// TIA Portal V20 export
TYPE "LBP_typeModeGroup"
TITLE = Mode group signals / Signaux groupe de modes de fonctionnement
// User data type for block LBP_ModeGroup [DB11] / Type de données utilisateur pour bloc LBP_ModeGroup [DB11]
   STRUCT
      A_AUTO : Bool;   // Operating mode AUTOMATIC / Mode AUTOMATIC
      A_MDA : Bool;   // Operating mode MDA / Mode MDA
      A_JOG : Bool;   // Operating mode JOG / Mode JOG
      f0_3 : Bool;
      A_MCDisable : Bool;   // Mode change disable / Désactiver changement mode de fonctionnement
      A_MGStop : Bool;   // Mode group stop / Groupe de modes de fonctionnement Arrêt
      A_MGStopASp : Bool;   // Mode group stop axes plus spindle / Groupe de modes de fonctionnement Arrêt axes et broche
      A_MGReset : Bool;   // Mode group reset / Groupe de modes de fonctionnement Reset
      A_TEACHIN : Bool;   // Machine function TEACH IN / Fonction machine TEACH IN
      A_REPOS : Bool;   // Machine function REPOS / Fonction machine REPOS
      A_REF : Bool;   // Machine function REF / Fonction machine REF
      f1_3 : Bool;
      f1_4 : Bool;
      f1_5 : Bool;
      A_SingleBlock_B : Bool;   // Single block type B / Bloc par bloc type B
      A_SingleBlock_A : Bool;   // Single block type A / Bloc par bloc type A
      A_INC1 : Bool;   // INC1
      A_INC10 : Bool;   // INC10
      A_INC100 : Bool;   // INC100
      A_INC1000 : Bool;   // INC1000
      A_INC10000 : Bool;   // INC10000
      A_INCVar : Bool;   // INC variable / Variable INC
      A_ContManTravel : Bool;   // Continuous manual travel / Mode manuel continu
      f2_7 : Bool;
      f3 : Byte;
      E_MMC_AUTO : Bool;   // HMI mode strobe AUTOMATIC / HMI mode Strobe AUTOMATIC
      E_MMC_MDA : Bool;   // HMI mode strobe MDA / HMI mode Strobe MDA
      E_MMC_JOG : Bool;   // HMI mode strobe JOG / HMI mode Strobe JOG
      f4_3 : Bool;
      f4_4 : Bool;
      f4_5 : Bool;
      f4_6 : Bool;
      f4_7 : Bool;
      E_MMC_TEACHIN : Bool;   // HMI machine function strobe TEACH IN / HMI Fonction machine Strobe TEACH IN
      E_MMC_REPOS : Bool;   // HMI machine function strobe REPOS / HMI Fonction machine Strobe REPOS
      E_MMC_REF : Bool;   // HMI machine function strobe REF / HMI Fonction machine Strobe REF
      f5_3 : Bool;
      f5_4 : Bool;
      f5_5 : Bool;
      f5_6 : Bool;
      f5_7 : Bool;
      E_AUTO : Bool;   // Active operating mode AUTOMATIC / Mode actif AUTOMATIC
      E_MDA : Bool;   // Active operating mode MDA / Mode actif MDA
      E_JOG : Bool;   // Active operating mode JOG / Mode actif JOG
      E_MGOK : Bool;   // Mode group ready / Groupe de modes de fonctionnement prêt
      E_MGreseted : Bool;   // Mode group reset performed / Groupe de modes de fonctionnement Reset effectué
      E_NCKintJOG : Bool;   // NCK internal JOG active / NCK JOG interne actif
      f6_6 : Bool;
      E_ChanReset : Bool;   // All channels in reset state / Tous les canaux en mode Reset
      E_TEACHIN : Bool;   // Active machine function TEACH IN / Fonction machine active TEACH IN
      E_REPOS : Bool;   // Active machine function REPOS / Fonction machine active REPOS
      E_REF : Bool;   // Active machine function REF / Fonction machine active REF
      f7_3 : Bool;
      f7_4 : Bool;
      f7_5 : Bool;
      f7_6 : Bool;
      f7_7 : Bool;
      E_INC1 : Bool;   // INC1
      E_INC10 : Bool;   // INC10
      E_INC100 : Bool;   // INC100
      E_INC1000 : Bool;   // INC1000
      E_INC10000 : Bool;   // INC10000
      E_INCVar : Bool;   // INC variable / Variable INC
      E_ContManTravelAct : Bool;   // Continuous manual travel active / Mode manuel continu actif
      f8_7 : Bool;
      f9 : Byte;
      E_HMI_INC1 : Bool;   // INC1 from HMI / INC1 depuis IHM
      E_HMI_INC10 : Bool;   // INC10 from HMI / INC10 depuis IHM
      E_HMI_INC100 : Bool;   // INC100 from HMI / INC100 depuis IHM
      E_HMI_INC1000 : Bool;   // INC1000 from HMI / INC1000 depuis IHM
      E_HMI_INC10000 : Bool;   // INC10000 from HMI / INC10000 depuis IHM
      E_HMI_INCVar : Bool;   // INC variable from HMI / Variable INC depuis IHM
      E_HMI_ContManTravel : Bool;   // Continuous manual travel active from HMI / Course manuelle continue active depuis IHM
      f10_7 : Bool;
      f11 : Byte;
      f12 : Array[12..19] of Byte;
      MG : Array[2..10] of Struct   // next mode group from DBB20, as before / groupe de mode suivant depuis DBB20, comme avant
         A_AUTO : Bool;   // Operating mode AUTOMATIC / Mode AUTOMATIC
         A_MDA : Bool;   // Operating mode MDA / Mode MDA
         A_JOG : Bool;   // Operating mode JOG / Mode JOG
         f0_3 : Bool;
         A_MCDisable : Bool;   // Mode change disable / Désactiver changement mode de fonctionnement
         A_MGStop : Bool;   // Mode group stop / Groupe de modes de fonctionnement Arrêt
         A_MGStopASp : Bool;   // Mode group stop axes plus spindle / Groupe de modes de fonctionnement Arrêt axes et broche
         A_MGReset : Bool;   // Mode group reset / Groupe de modes de fonctionnement Reset
         A_TEACHIN : Bool;   // Machine function TEACH IN / Fonction machine TEACH IN
         A_REPOS : Bool;   // Machine function REPOS / Fonction machine REPOS
         A_REF : Bool;   // Machine function REF / Fonction machine REF
         f1_3 : Bool;
         f1_4 : Bool;
         f1_5 : Bool;
         A_SingleBlock_B : Bool;   // Single block type B / Bloc par bloc type B
         A_SingleBlock_A : Bool;   // Single block type A / Bloc par bloc type A
         A_INC1 : Bool;   // INC1
         A_INC10 : Bool;   // INC10
         A_INC100 : Bool;   // INC100
         A_INC1000 : Bool;   // INC1000
         A_INC10000 : Bool;   // INC10000
         A_INCVar : Bool;   // INC variable / Variable INC
         A_ContManTravel : Bool;   // Continuous manual travel / Mode manuel continu
         f2_7 : Bool;
         f3 : Byte;
         E_MMC_AUTO : Bool;   // HMI mode strobe AUTOMATIC / HMI mode Strobe AUTOMATIC
         E_MMC_MDA : Bool;   // HMI mode strobe MDA / HMI mode Strobe MDA
         E_MMC_JOG : Bool;   // HMI mode strobe JOG / HMI mode Strobe JOG
         f4_3 : Bool;
         f4_4 : Bool;
         f4_5 : Bool;
         f4_6 : Bool;
         f4_7 : Bool;
         E_MMC_TEACHIN : Bool;   // HMI machine function strobe TEACH IN / HMI Fonction machine Strobe TEACH IN
         E_MMC_REPOS : Bool;   // HMI machine function strobe REPOS / HMI Fonction machine Strobe REPOS
         E_MMC_REF : Bool;   // HMI machine function strobe REF / HMI Fonction machine Strobe REF
         f5_3 : Bool;
         f5_4 : Bool;
         f5_5 : Bool;
         f5_6 : Bool;
         f5_7 : Bool;
         E_AUTO : Bool;   // Active operating mode AUTOMATIC / Mode actif AUTOMATIC
         E_MDA : Bool;   // Active operating mode MDA / Mode actif MDA
         E_JOG : Bool;   // Active operating mode JOG / Mode actif JOG
         E_MGOK : Bool;   // Mode group ready / Groupe de modes de fonctionnement prêt
         E_MGreseted : Bool;   // Mode group reset / Groupe de modes de fonctionnement Reset
         E_NCKintJOG : Bool;   // NCK internal JOG active / NCK JOG interne actif
         f6_6 : Bool;
         E_ChanReset : Bool;   // All channels in reset state / Tous les canaux en mode Reset
         E_TEACHIN : Bool;   // Active machine function TEACH IN / Fonction machine active TEACH IN
         E_REPOS : Bool;   // Active machine function REPOS / Fonction machine active REPOS
         E_REF : Bool;   // Active machine function REF / Fonction machine active REF
         f7_3 : Bool;
         f7_4 : Bool;
         f7_5 : Bool;
         f7_6 : Bool;
         f7_7 : Bool;
         E_INC1 : Bool;   // INC1
         E_INC10 : Bool;   // INC10
         E_INC100 : Bool;   // INC100
         E_INC1000 : Bool;   // INC1000
         E_INC10000 : Bool;   // INC10000
         E_INCVar : Bool;   // INC variable / Variable INC
         E_ContManTravelAct : Bool;   // Continuous manual travel active / Mode manuel continu actif
         f8_7 : Bool;
         f9 : Byte;
         E_HMI_INC1 : Bool;   // INC1 from HMI / INC1 depuis IHM
         E_HMI_INC10 : Bool;   // INC10 from HMI / INC10 depuis IHM
         E_HMI_INC100 : Bool;   // INC100 from HMI / INC100 depuis IHM
         E_HMI_INC1000 : Bool;   // INC1000 from HMI / INC1000 depuis IHM
         E_HMI_INC10000 : Bool;   // INC10000 from HMI / INC10000 depuis IHM
         E_HMI_INCVar : Bool;   // INC variable from HMI / Variable INC depuis IHM
         E_HMI_ContManTravel : Bool;   // Continuous manual travel active from HMI / Course manuelle continue active depuis IHM
         f10_7 : Bool;
         f11 : Byte;
         f12 : Array[12..19] of Byte;
      END_STRUCT;
   END_STRUCT;
   // // MG[3].A_AUTO : Operating mode AUTOMATIC / Mode AUTOMATIC
   // // MG[4].A_AUTO : Operating mode AUTOMATIC / Mode AUTOMATIC
   // // MG[5].A_AUTO : Operating mode AUTOMATIC / Mode AUTOMATIC
   // // MG[6].A_AUTO : Operating mode AUTOMATIC / Mode AUTOMATIC
   // // MG[7].A_AUTO : Operating mode AUTOMATIC / Mode AUTOMATIC
   // // MG[8].A_AUTO : Operating mode AUTOMATIC / Mode AUTOMATIC
   // // MG[9].A_AUTO : Operating mode AUTOMATIC / Mode AUTOMATIC
   // // MG[10].A_AUTO : Operating mode AUTOMATIC / Mode AUTOMATIC
   // // MG[3].A_MDA : Operating mode MDA / Mode MDA
   // // MG[4].A_MDA : Operating mode MDA / Mode MDA
   // // MG[5].A_MDA : Operating mode MDA / Mode MDA
   // // MG[6].A_MDA : Operating mode MDA / Mode MDA
   // // MG[7].A_MDA : Operating mode MDA / Mode MDA
   // // MG[8].A_MDA : Operating mode MDA / Mode MDA
   // // MG[9].A_MDA : Operating mode MDA / Mode MDA
   // // MG[10].A_MDA : Operating mode MDA / Mode MDA
   // // MG[3].A_JOG : Operating mode JOG / Mode JOG
   // // MG[4].A_JOG : Operating mode JOG / Mode JOG
   // // MG[5].A_JOG : Operating mode JOG / Mode JOG
   // // MG[6].A_JOG : Operating mode JOG / Mode JOG
   // // MG[7].A_JOG : Operating mode JOG / Mode JOG
   // // MG[8].A_JOG : Operating mode JOG / Mode JOG
   // // MG[9].A_JOG : Operating mode JOG / Mode JOG
   // // MG[10].A_JOG : Operating mode JOG / Mode JOG
   // // MG[3].A_MCDisable : Mode change disable / Désactiver changement mode de fonctionnement
   // // MG[4].A_MCDisable : Mode change disable / Désactiver changement mode de fonctionnement
   // // MG[5].A_MCDisable : Mode change disable / Désactiver changement mode de fonctionnement
   // // MG[6].A_MCDisable : Mode change disable / Désactiver changement mode de fonctionnement
   // // MG[7].A_MCDisable : Mode change disable / Désactiver changement mode de fonctionnement
   // // MG[8].A_MCDisable : Mode change disable / Désactiver changement mode de fonctionnement
   // // MG[9].A_MCDisable : Mode change disable / Désactiver changement mode de fonctionnement
   // // MG[10].A_MCDisable : Mode change disable / Désactiver changement mode de fonctionnement
   // // MG[3].A_MGStop : Mode group stop / Groupe de modes de fonctionnement Arrêt
   // // MG[4].A_MGStop : Mode group stop / Groupe de modes de fonctionnement Arrêt
   // // MG[5].A_MGStop : Mode group stop / Groupe de modes de fonctionnement Arrêt
   // // MG[6].A_MGStop : Mode group stop / Groupe de modes de fonctionnement Arrêt
   // // MG[7].A_MGStop : Mode group stop / Groupe de modes de fonctionnement Arrêt
   // // MG[8].A_MGStop : Mode group stop / Groupe de modes de fonctionnement Arrêt
   // // MG[9].A_MGStop : Mode group stop / Groupe de modes de fonctionnement Arrêt
   // // MG[10].A_MGStop : Mode group stop / Groupe de modes de fonctionnement Arrêt
   // // MG[3].A_MGStopASp : Mode group stop axes plus spindle / Groupe de modes de fonctionnement Arrêt axes et broche
   // // MG[4].A_MGStopASp : Mode group stop axes plus spindle / Groupe de modes de fonctionnement Arrêt axes et broche
   // // MG[5].A_MGStopASp : Mode group stop axes plus spindle / Groupe de modes de fonctionnement Arrêt axes et broche
   // // MG[6].A_MGStopASp : Mode group stop axes plus spindle / Groupe de modes de fonctionnement Arrêt axes et broche
   // // MG[7].A_MGStopASp : Mode group stop axes plus spindle / Groupe de modes de fonctionnement Arrêt axes et broche
   // // MG[8].A_MGStopASp : Mode group stop axes plus spindle / Groupe de modes de fonctionnement Arrêt axes et broche
   // // MG[9].A_MGStopASp : Mode group stop axes plus spindle / Groupe de modes de fonctionnement Arrêt axes et broche
   // // MG[10].A_MGStopASp : Mode group stop axes plus spindle / Groupe de modes de fonctionnement Arrêt axes et broche
   // // MG[3].A_MGReset : Mode group reset / Groupe de modes de fonctionnement Reset
   // // MG[4].A_MGReset : Mode group reset / Groupe de modes de fonctionnement Reset
   // // MG[5].A_MGReset : Mode group reset / Groupe de modes de fonctionnement Reset
   // // MG[6].A_MGReset : Mode group reset / Groupe de modes de fonctionnement Reset
   // // MG[7].A_MGReset : Mode group reset / Groupe de modes de fonctionnement Reset
   // // MG[8].A_MGReset : Mode group reset / Groupe de modes de fonctionnement Reset
   // // MG[9].A_MGReset : Mode group reset / Groupe de modes de fonctionnement Reset
   // // MG[10].A_MGReset : Mode group reset / Groupe de modes de fonctionnement Reset
   // // MG[3].A_TEACHIN : Machine function TEACH IN / Fonction machine TEACH IN
   // // MG[4].A_TEACHIN : Machine function TEACH IN / Fonction machine TEACH IN
   // // MG[5].A_TEACHIN : Machine function TEACH IN / Fonction machine TEACH IN
   // // MG[6].A_TEACHIN : Machine function TEACH IN / Fonction machine TEACH IN
   // // MG[7].A_TEACHIN : Machine function TEACH IN / Fonction machine TEACH IN
   // // MG[8].A_TEACHIN : Machine function TEACH IN / Fonction machine TEACH IN
   // // MG[9].A_TEACHIN : Machine function TEACH IN / Fonction machine TEACH IN
   // // MG[10].A_TEACHIN : Machine function TEACH IN / Fonction machine TEACH IN
   // // MG[3].A_REPOS : Machine function REPOS / Fonction machine REPOS
   // // MG[4].A_REPOS : Machine function REPOS / Fonction machine REPOS
   // // MG[5].A_REPOS : Machine function REPOS / Fonction machine REPOS
   // // MG[6].A_REPOS : Machine function REPOS / Fonction machine REPOS
   // // MG[7].A_REPOS : Machine function REPOS / Fonction machine REPOS
   // // MG[8].A_REPOS : Machine function REPOS / Fonction machine REPOS
   // // MG[9].A_REPOS : Machine function REPOS / Fonction machine REPOS
   // // MG[10].A_REPOS : Machine function REPOS / Fonction machine REPOS
   // // MG[3].A_REF : Machine function REF / Fonction machine REF
   // // MG[4].A_REF : Machine function REF / Fonction machine REF
   // // MG[5].A_REF : Machine function REF / Fonction machine REF
   // // MG[6].A_REF : Machine function REF / Fonction machine REF
   // // MG[7].A_REF : Machine function REF / Fonction machine REF
   // // MG[8].A_REF : Machine function REF / Fonction machine REF
   // // MG[9].A_REF : Machine function REF / Fonction machine REF
   // // MG[10].A_REF : Machine function REF / Fonction machine REF
   // // MG[3].A_SingleBlock_B : Single block type B / Bloc par bloc type B
   // // MG[4].A_SingleBlock_B : Single block type B / Bloc par bloc type B
   // // MG[5].A_SingleBlock_B : Single block type B / Bloc par bloc type B
   // // MG[6].A_SingleBlock_B : Single block type B / Bloc par bloc type B
   // // MG[7].A_SingleBlock_B : Single block type B / Bloc par bloc type B
   // // MG[8].A_SingleBlock_B : Single block type B / Bloc par bloc type B
   // // MG[9].A_SingleBlock_B : Single block type B / Bloc par bloc type B
   // // MG[10].A_SingleBlock_B : Single block type B / Bloc par bloc type B
   // // MG[3].A_SingleBlock_A : Single block type A / Bloc par bloc type A
   // // MG[4].A_SingleBlock_A : Single block type A / Bloc par bloc type A
   // // MG[5].A_SingleBlock_A : Single block type A / Bloc par bloc type A
   // // MG[6].A_SingleBlock_A : Single block type A / Bloc par bloc type A
   // // MG[7].A_SingleBlock_A : Single block type A / Bloc par bloc type A
   // // MG[8].A_SingleBlock_A : Single block type A / Bloc par bloc type A
   // // MG[9].A_SingleBlock_A : Single block type A / Bloc par bloc type A
   // // MG[10].A_SingleBlock_A : Single block type A / Bloc par bloc type A
   // // MG[3].A_INC1 : INC1
   // // MG[4].A_INC1 : INC1
   // // MG[5].A_INC1 : INC1
   // // MG[6].A_INC1 : INC1
   // // MG[7].A_INC1 : INC1
   // // MG[8].A_INC1 : INC1
   // // MG[9].A_INC1 : INC1
   // // MG[10].A_INC1 : INC1
   // // MG[3].A_INC10 : INC10
   // // MG[4].A_INC10 : INC10
   // // MG[5].A_INC10 : INC10
   // // MG[6].A_INC10 : INC10
   // // MG[7].A_INC10 : INC10
   // // MG[8].A_INC10 : INC10
   // // MG[9].A_INC10 : INC10
   // // MG[10].A_INC10 : INC10
   // // MG[3].A_INC100 : INC100
   // // MG[4].A_INC100 : INC100
   // // MG[5].A_INC100 : INC100
   // // MG[6].A_INC100 : INC100
   // // MG[7].A_INC100 : INC100
   // // MG[8].A_INC100 : INC100
   // // MG[9].A_INC100 : INC100
   // // MG[10].A_INC100 : INC100
   // // MG[3].A_INC1000 : INC1000
   // // MG[4].A_INC1000 : INC1000
   // // MG[5].A_INC1000 : INC1000
   // // MG[6].A_INC1000 : INC1000
   // // MG[7].A_INC1000 : INC1000
   // // MG[8].A_INC1000 : INC1000
   // // MG[9].A_INC1000 : INC1000
   // // MG[10].A_INC1000 : INC1000
   // // MG[3].A_INC10000 : INC10000
   // // MG[4].A_INC10000 : INC10000
   // // MG[5].A_INC10000 : INC10000
   // // MG[6].A_INC10000 : INC10000
   // // MG[7].A_INC10000 : INC10000
   // // MG[8].A_INC10000 : INC10000
   // // MG[9].A_INC10000 : INC10000
   // // MG[10].A_INC10000 : INC10000
   // // MG[3].A_INCVar : INC variable / Variable INC
   // // MG[4].A_INCVar : INC variable / Variable INC
   // // MG[5].A_INCVar : INC variable / Variable INC
   // // MG[6].A_INCVar : INC variable / Variable INC
   // // MG[7].A_INCVar : INC variable / Variable INC
   // // MG[8].A_INCVar : INC variable / Variable INC
   // // MG[9].A_INCVar : INC variable / Variable INC
   // // MG[10].A_INCVar : INC variable / Variable INC
   // // MG[3].A_ContManTravel : Continuous manual travel / Mode manuel continu
   // // MG[4].A_ContManTravel : Continuous manual travel / Mode manuel continu
   // // MG[5].A_ContManTravel : Continuous manual travel / Mode manuel continu
   // // MG[6].A_ContManTravel : Continuous manual travel / Mode manuel continu
   // // MG[7].A_ContManTravel : Continuous manual travel / Mode manuel continu
   // // MG[8].A_ContManTravel : Continuous manual travel / Mode manuel continu
   // // MG[9].A_ContManTravel : Continuous manual travel / Mode manuel continu
   // // MG[10].A_ContManTravel : Continuous manual travel / Mode manuel continu
   // // MG[3].E_MMC_AUTO : HMI mode strobe AUTOMATIC / HMI mode Strobe AUTOMATIC
   // // MG[4].E_MMC_AUTO : HMI mode strobe AUTOMATIC / HMI mode Strobe AUTOMATIC
   // // MG[5].E_MMC_AUTO : HMI mode strobe AUTOMATIC / HMI mode Strobe AUTOMATIC
   // // MG[6].E_MMC_AUTO : HMI mode strobe AUTOMATIC / HMI mode Strobe AUTOMATIC
   // // MG[7].E_MMC_AUTO : HMI mode strobe AUTOMATIC / HMI mode Strobe AUTOMATIC
   // // MG[8].E_MMC_AUTO : HMI mode strobe AUTOMATIC / HMI mode Strobe AUTOMATIC
   // // MG[9].E_MMC_AUTO : HMI mode strobe AUTOMATIC / HMI mode Strobe AUTOMATIC
   // // MG[10].E_MMC_AUTO : HMI mode strobe AUTOMATIC / HMI mode Strobe AUTOMATIC
   // // MG[3].E_MMC_MDA : HMI mode strobe MDA / HMI mode Strobe MDA
   // // MG[4].E_MMC_MDA : HMI mode strobe MDA / HMI mode Strobe MDA
   // // MG[5].E_MMC_MDA : HMI mode strobe MDA / HMI mode Strobe MDA
   // // MG[6].E_MMC_MDA : HMI mode strobe MDA / HMI mode Strobe MDA
   // // MG[7].E_MMC_MDA : HMI mode strobe MDA / HMI mode Strobe MDA
   // // MG[8].E_MMC_MDA : HMI mode strobe MDA / HMI mode Strobe MDA
   // // MG[9].E_MMC_MDA : HMI mode strobe MDA / HMI mode Strobe MDA
   // // MG[10].E_MMC_MDA : HMI mode strobe MDA / HMI mode Strobe MDA
   // // MG[3].E_MMC_JOG : HMI mode strobe JOG / HMI mode Strobe JOG
   // // MG[4].E_MMC_JOG : HMI mode strobe JOG / HMI mode Strobe JOG
   // // MG[5].E_MMC_JOG : HMI mode strobe JOG / HMI mode Strobe JOG
   // // MG[6].E_MMC_JOG : HMI mode strobe JOG / HMI mode Strobe JOG
   // // MG[7].E_MMC_JOG : HMI mode strobe JOG / HMI mode Strobe JOG
   // // MG[8].E_MMC_JOG : HMI mode strobe JOG / HMI mode Strobe JOG
   // // MG[9].E_MMC_JOG : HMI mode strobe JOG / HMI mode Strobe JOG
   // // MG[10].E_MMC_JOG : HMI mode strobe JOG / HMI mode Strobe JOG
   // // MG[3].E_MMC_TEACHIN : HMI machine function strobe TEACH IN / HMI Fonction machine Strobe TEACH IN
   // // MG[4].E_MMC_TEACHIN : HMI machine function strobe TEACH IN / HMI Fonction machine Strobe TEACH IN
   // // MG[5].E_MMC_TEACHIN : HMI machine function strobe TEACH IN / HMI Fonction machine Strobe TEACH IN
   // // MG[6].E_MMC_TEACHIN : HMI machine function strobe TEACH IN / HMI Fonction machine Strobe TEACH IN
   // // MG[7].E_MMC_TEACHIN : HMI machine function strobe TEACH IN / HMI Fonction machine Strobe TEACH IN
   // // MG[8].E_MMC_TEACHIN : HMI machine function strobe TEACH IN / HMI Fonction machine Strobe TEACH IN
   // // MG[9].E_MMC_TEACHIN : HMI machine function strobe TEACH IN / HMI Fonction machine Strobe TEACH IN
   // // MG[10].E_MMC_TEACHIN : HMI machine function strobe TEACH IN / HMI Fonction machine Strobe TEACH IN
   // // MG[3].E_MMC_REPOS : HMI machine function strobe REPOS / HMI Fonction machine Strobe REPOS
   // // MG[4].E_MMC_REPOS : HMI machine function strobe REPOS / HMI Fonction machine Strobe REPOS
   // // MG[5].E_MMC_REPOS : HMI machine function strobe REPOS / HMI Fonction machine Strobe REPOS
   // // MG[6].E_MMC_REPOS : HMI machine function strobe REPOS / HMI Fonction machine Strobe REPOS
   // // MG[7].E_MMC_REPOS : HMI machine function strobe REPOS / HMI Fonction machine Strobe REPOS
   // // MG[8].E_MMC_REPOS : HMI machine function strobe REPOS / HMI Fonction machine Strobe REPOS
   // // MG[9].E_MMC_REPOS : HMI machine function strobe REPOS / HMI Fonction machine Strobe REPOS
   // // MG[10].E_MMC_REPOS : HMI machine function strobe REPOS / HMI Fonction machine Strobe REPOS
   // // MG[3].E_MMC_REF : HMI machine function strobe REF / HMI Fonction machine Strobe REF
   // // MG[4].E_MMC_REF : HMI machine function strobe REF / HMI Fonction machine Strobe REF
   // // MG[5].E_MMC_REF : HMI machine function strobe REF / HMI Fonction machine Strobe REF
   // // MG[6].E_MMC_REF : HMI machine function strobe REF / HMI Fonction machine Strobe REF
   // // MG[7].E_MMC_REF : HMI machine function strobe REF / HMI Fonction machine Strobe REF
   // // MG[8].E_MMC_REF : HMI machine function strobe REF / HMI Fonction machine Strobe REF
   // // MG[9].E_MMC_REF : HMI machine function strobe REF / HMI Fonction machine Strobe REF
   // // MG[10].E_MMC_REF : HMI machine function strobe REF / HMI Fonction machine Strobe REF
   // // MG[3].E_AUTO : Active operating mode AUTOMATIC / Mode actif AUTOMATIC
   // // MG[4].E_AUTO : Active operating mode AUTOMATIC / Mode actif AUTOMATIC
   // // MG[5].E_AUTO : Active operating mode AUTOMATIC / Mode actif AUTOMATIC
   // // MG[6].E_AUTO : Active operating mode AUTOMATIC / Mode actif AUTOMATIC
   // // MG[7].E_AUTO : Active operating mode AUTOMATIC / Mode actif AUTOMATIC
   // // MG[8].E_AUTO : Active operating mode AUTOMATIC / Mode actif AUTOMATIC
   // // MG[9].E_AUTO : Active operating mode AUTOMATIC / Mode actif AUTOMATIC
   // // MG[10].E_AUTO : Active operating mode AUTOMATIC / Mode actif AUTOMATIC
   // // MG[3].E_MDA : Active operating mode MDA / Mode actif MDA
   // // MG[4].E_MDA : Active operating mode MDA / Mode actif MDA
   // // MG[5].E_MDA : Active operating mode MDA / Mode actif MDA
   // // MG[6].E_MDA : Active operating mode MDA / Mode actif MDA
   // // MG[7].E_MDA : Active operating mode MDA / Mode actif MDA
   // // MG[8].E_MDA : Active operating mode MDA / Mode actif MDA
   // // MG[9].E_MDA : Active operating mode MDA / Mode actif MDA
   // // MG[10].E_MDA : Active operating mode MDA / Mode actif MDA
   // // MG[3].E_JOG : Active operating mode JOG / Mode actif JOG
   // // MG[4].E_JOG : Active operating mode JOG / Mode actif JOG
   // // MG[5].E_JOG : Active operating mode JOG / Mode actif JOG
   // // MG[6].E_JOG : Active operating mode JOG / Mode actif JOG
   // // MG[7].E_JOG : Active operating mode JOG / Mode actif JOG
   // // MG[8].E_JOG : Active operating mode JOG / Mode actif JOG
   // // MG[9].E_JOG : Active operating mode JOG / Mode actif JOG
   // // MG[10].E_JOG : Active operating mode JOG / Mode actif JOG
   // // MG[3].E_MGOK : Mode group ready / Groupe de modes de fonctionnement prêt
   // // MG[4].E_MGOK : Mode group ready / Groupe de modes de fonctionnement prêt
   // // MG[5].E_MGOK : Mode group ready / Groupe de modes de fonctionnement prêt
   // // MG[6].E_MGOK : Mode group ready / Groupe de modes de fonctionnement prêt
   // // MG[7].E_MGOK : Mode group ready / Groupe de modes de fonctionnement prêt
   // // MG[8].E_MGOK : Mode group ready / Groupe de modes de fonctionnement prêt
   // // MG[9].E_MGOK : Mode group ready / Groupe de modes de fonctionnement prêt
   // // MG[10].E_MGOK : Mode group ready / Groupe de modes de fonctionnement prêt
   // // MG[3].E_MGreseted : Mode group reset / Groupe de modes de fonctionnement Reset
   // // MG[4].E_MGreseted : Mode group reset / Groupe de modes de fonctionnement Reset
   // // MG[5].E_MGreseted : Mode group reset / Groupe de modes de fonctionnement Reset
   // // MG[6].E_MGreseted : Mode group reset / Groupe de modes de fonctionnement Reset
   // // MG[7].E_MGreseted : Mode group reset / Groupe de modes de fonctionnement Reset
   // // MG[8].E_MGreseted : Mode group reset / Groupe de modes de fonctionnement Reset
   // // MG[9].E_MGreseted : Mode group reset / Groupe de modes de fonctionnement Reset
   // // MG[10].E_MGreseted : Mode group reset / Groupe de modes de fonctionnement Reset
   // // MG[3].E_NCKintJOG : NCK internal JOG active / NCK JOG interne actif
   // // MG[4].E_NCKintJOG : NCK internal JOG active / NCK JOG interne actif
   // // MG[5].E_NCKintJOG : NCK internal JOG active / NCK JOG interne actif
   // // MG[6].E_NCKintJOG : NCK internal JOG active / NCK JOG interne actif
   // // MG[7].E_NCKintJOG : NCK internal JOG active / NCK JOG interne actif
   // // MG[8].E_NCKintJOG : NCK internal JOG active / NCK JOG interne actif
   // // MG[9].E_NCKintJOG : NCK internal JOG active / NCK JOG interne actif
   // // MG[10].E_NCKintJOG : NCK internal JOG active / NCK JOG interne actif
   // // MG[3].E_ChanReset : All channels in reset state / Tous les canaux en mode Reset
   // // MG[4].E_ChanReset : All channels in reset state / Tous les canaux en mode Reset
   // // MG[5].E_ChanReset : All channels in reset state / Tous les canaux en mode Reset
   // // MG[6].E_ChanReset : All channels in reset state / Tous les canaux en mode Reset
   // // MG[7].E_ChanReset : All channels in reset state / Tous les canaux en mode Reset
   // // MG[8].E_ChanReset : All channels in reset state / Tous les canaux en mode Reset
   // // MG[9].E_ChanReset : All channels in reset state / Tous les canaux en mode Reset
   // // MG[10].E_ChanReset : All channels in reset state / Tous les canaux en mode Reset
   // // MG[3].E_TEACHIN : Active machine function TEACH IN / Fonction machine active TEACH IN
   // // MG[4].E_TEACHIN : Active machine function TEACH IN / Fonction machine active TEACH IN
   // // MG[5].E_TEACHIN : Active machine function TEACH IN / Fonction machine active TEACH IN
   // // MG[6].E_TEACHIN : Active machine function TEACH IN / Fonction machine active TEACH IN
   // // MG[7].E_TEACHIN : Active machine function TEACH IN / Fonction machine active TEACH IN
   // // MG[8].E_TEACHIN : Active machine function TEACH IN / Fonction machine active TEACH IN
   // // MG[9].E_TEACHIN : Active machine function TEACH IN / Fonction machine active TEACH IN
   // // MG[10].E_TEACHIN : Active machine function TEACH IN / Fonction machine active TEACH IN
   // // MG[3].E_REPOS : Active machine function REPOS / Fonction machine active REPOS
   // // MG[4].E_REPOS : Active machine function REPOS / Fonction machine active REPOS
   // // MG[5].E_REPOS : Active machine function REPOS / Fonction machine active REPOS
   // // MG[6].E_REPOS : Active machine function REPOS / Fonction machine active REPOS
   // // MG[7].E_REPOS : Active machine function REPOS / Fonction machine active REPOS
   // // MG[8].E_REPOS : Active machine function REPOS / Fonction machine active REPOS
   // // MG[9].E_REPOS : Active machine function REPOS / Fonction machine active REPOS
   // // MG[10].E_REPOS : Active machine function REPOS / Fonction machine active REPOS
   // // MG[3].E_REF : Active machine function REF / Fonction machine active REF
   // // MG[4].E_REF : Active machine function REF / Fonction machine active REF
   // // MG[5].E_REF : Active machine function REF / Fonction machine active REF
   // // MG[6].E_REF : Active machine function REF / Fonction machine active REF
   // // MG[7].E_REF : Active machine function REF / Fonction machine active REF
   // // MG[8].E_REF : Active machine function REF / Fonction machine active REF
   // // MG[9].E_REF : Active machine function REF / Fonction machine active REF
   // // MG[10].E_REF : Active machine function REF / Fonction machine active REF
   // // MG[3].E_INC1 : INC1
   // // MG[4].E_INC1 : INC1
   // // MG[5].E_INC1 : INC1
   // // MG[6].E_INC1 : INC1
   // // MG[7].E_INC1 : INC1
   // // MG[8].E_INC1 : INC1
   // // MG[9].E_INC1 : INC1
   // // MG[10].E_INC1 : INC1
   // // MG[3].E_INC10 : INC10
   // // MG[4].E_INC10 : INC10
   // // MG[5].E_INC10 : INC10
   // // MG[6].E_INC10 : INC10
   // // MG[7].E_INC10 : INC10
   // // MG[8].E_INC10 : INC10
   // // MG[9].E_INC10 : INC10
   // // MG[10].E_INC10 : INC10
   // // MG[3].E_INC100 : INC100
   // // MG[4].E_INC100 : INC100
   // // MG[5].E_INC100 : INC100
   // // MG[6].E_INC100 : INC100
   // // MG[7].E_INC100 : INC100
   // // MG[8].E_INC100 : INC100
   // // MG[9].E_INC100 : INC100
   // // MG[10].E_INC100 : INC100
   // // MG[3].E_INC1000 : INC1000
   // // MG[4].E_INC1000 : INC1000
   // // MG[5].E_INC1000 : INC1000
   // // MG[6].E_INC1000 : INC1000
   // // MG[7].E_INC1000 : INC1000
   // // MG[8].E_INC1000 : INC1000
   // // MG[9].E_INC1000 : INC1000
   // // MG[10].E_INC1000 : INC1000
   // // MG[3].E_INC10000 : INC10000
   // // MG[4].E_INC10000 : INC10000
   // // MG[5].E_INC10000 : INC10000
   // // MG[6].E_INC10000 : INC10000
   // // MG[7].E_INC10000 : INC10000
   // // MG[8].E_INC10000 : INC10000
   // // MG[9].E_INC10000 : INC10000
   // // MG[10].E_INC10000 : INC10000
   // // MG[3].E_INCVar : INC variable / Variable INC
   // // MG[4].E_INCVar : INC variable / Variable INC
   // // MG[5].E_INCVar : INC variable / Variable INC
   // // MG[6].E_INCVar : INC variable / Variable INC
   // // MG[7].E_INCVar : INC variable / Variable INC
   // // MG[8].E_INCVar : INC variable / Variable INC
   // // MG[9].E_INCVar : INC variable / Variable INC
   // // MG[10].E_INCVar : INC variable / Variable INC
   // // MG[3].E_ContManTravelAct : Continuous manual travel active / Mode manuel continu actif
   // // MG[4].E_ContManTravelAct : Continuous manual travel active / Mode manuel continu actif
   // // MG[5].E_ContManTravelAct : Continuous manual travel active / Mode manuel continu actif
   // // MG[6].E_ContManTravelAct : Continuous manual travel active / Mode manuel continu actif
   // // MG[7].E_ContManTravelAct : Continuous manual travel active / Mode manuel continu actif
   // // MG[8].E_ContManTravelAct : Continuous manual travel active / Mode manuel continu actif
   // // MG[9].E_ContManTravelAct : Continuous manual travel active / Mode manuel continu actif
   // // MG[10].E_ContManTravelAct : Continuous manual travel active / Mode manuel continu actif
   // // MG[3].E_HMI_INC1 : INC1 from HMI / INC1 depuis IHM
   // // MG[4].E_HMI_INC1 : INC1 from HMI / INC1 depuis IHM
   // // MG[5].E_HMI_INC1 : INC1 from HMI / INC1 depuis IHM
   // // MG[6].E_HMI_INC1 : INC1 from HMI / INC1 depuis IHM
   // // MG[7].E_HMI_INC1 : INC1 from HMI / INC1 depuis IHM
   // // MG[8].E_HMI_INC1 : INC1 from HMI / INC1 depuis IHM
   // // MG[9].E_HMI_INC1 : INC1 from HMI / INC1 depuis IHM
   // // MG[10].E_HMI_INC1 : INC1 from HMI / INC1 depuis IHM
   // // MG[3].E_HMI_INC10 : INC10 from HMI / INC10 depuis IHM
   // // MG[4].E_HMI_INC10 : INC10 from HMI / INC10 depuis IHM
   // // MG[5].E_HMI_INC10 : INC10 from HMI / INC10 depuis IHM
   // // MG[6].E_HMI_INC10 : INC10 from HMI / INC10 depuis IHM
   // // MG[7].E_HMI_INC10 : INC10 from HMI / INC10 depuis IHM
   // // MG[8].E_HMI_INC10 : INC10 from HMI / INC10 depuis IHM
   // // MG[9].E_HMI_INC10 : INC10 from HMI / INC10 depuis IHM
   // // MG[10].E_HMI_INC10 : INC10 from HMI / INC10 depuis IHM
   // // MG[3].E_HMI_INC100 : INC100 from HMI / INC100 depuis IHM
   // // MG[4].E_HMI_INC100 : INC100 from HMI / INC100 depuis IHM
   // // MG[5].E_HMI_INC100 : INC100 from HMI / INC100 depuis IHM
   // // MG[6].E_HMI_INC100 : INC100 from HMI / INC100 depuis IHM
   // // MG[7].E_HMI_INC100 : INC100 from HMI / INC100 depuis IHM
   // // MG[8].E_HMI_INC100 : INC100 from HMI / INC100 depuis IHM
   // // MG[9].E_HMI_INC100 : INC100 from HMI / INC100 depuis IHM
   // // MG[10].E_HMI_INC100 : INC100 from HMI / INC100 depuis IHM
   // // MG[3].E_HMI_INC1000 : INC1000 from HMI / INC1000 depuis IHM
   // // MG[4].E_HMI_INC1000 : INC1000 from HMI / INC1000 depuis IHM
   // // MG[5].E_HMI_INC1000 : INC1000 from HMI / INC1000 depuis IHM
   // // MG[6].E_HMI_INC1000 : INC1000 from HMI / INC1000 depuis IHM
   // // MG[7].E_HMI_INC1000 : INC1000 from HMI / INC1000 depuis IHM
   // // MG[8].E_HMI_INC1000 : INC1000 from HMI / INC1000 depuis IHM
   // // MG[9].E_HMI_INC1000 : INC1000 from HMI / INC1000 depuis IHM
   // // MG[10].E_HMI_INC1000 : INC1000 from HMI / INC1000 depuis IHM
   // // MG[3].E_HMI_INC10000 : INC10000 from HMI / INC10000 depuis IHM
   // // MG[4].E_HMI_INC10000 : INC10000 from HMI / INC10000 depuis IHM
   // // MG[5].E_HMI_INC10000 : INC10000 from HMI / INC10000 depuis IHM
   // // MG[6].E_HMI_INC10000 : INC10000 from HMI / INC10000 depuis IHM
   // // MG[7].E_HMI_INC10000 : INC10000 from HMI / INC10000 depuis IHM
   // // MG[8].E_HMI_INC10000 : INC10000 from HMI / INC10000 depuis IHM
   // // MG[9].E_HMI_INC10000 : INC10000 from HMI / INC10000 depuis IHM
   // // MG[10].E_HMI_INC10000 : INC10000 from HMI / INC10000 depuis IHM
   // // MG[3].E_HMI_INCVar : INC variable from HMI / Variable INC depuis IHM
   // // MG[4].E_HMI_INCVar : INC variable from HMI / Variable INC depuis IHM
   // // MG[5].E_HMI_INCVar : INC variable from HMI / Variable INC depuis IHM
   // // MG[6].E_HMI_INCVar : INC variable from HMI / Variable INC depuis IHM
   // // MG[7].E_HMI_INCVar : INC variable from HMI / Variable INC depuis IHM
   // // MG[8].E_HMI_INCVar : INC variable from HMI / Variable INC depuis IHM
   // // MG[9].E_HMI_INCVar : INC variable from HMI / Variable INC depuis IHM
   // // MG[10].E_HMI_INCVar : INC variable from HMI / Variable INC depuis IHM
   // // MG[3].E_HMI_ContManTravel : Continuous manual travel active from HMI / Course manuelle continue active depuis IHM
   // // MG[4].E_HMI_ContManTravel : Continuous manual travel active from HMI / Course manuelle continue active depuis IHM
   // // MG[5].E_HMI_ContManTravel : Continuous manual travel active from HMI / Course manuelle continue active depuis IHM
   // // MG[6].E_HMI_ContManTravel : Continuous manual travel active from HMI / Course manuelle continue active depuis IHM
   // // MG[7].E_HMI_ContManTravel : Continuous manual travel active from HMI / Course manuelle continue active depuis IHM
   // // MG[8].E_HMI_ContManTravel : Continuous manual travel active from HMI / Course manuelle continue active depuis IHM
   // // MG[9].E_HMI_ContManTravel : Continuous manual travel active from HMI / Course manuelle continue active depuis IHM
   // // MG[10].E_HMI_ContManTravel : Continuous manual travel active from HMI / Course manuelle continue active depuis IHM
   // // MG[2] : next mode group from DBB20, as before / groupe de mode suivant depuis DBB20, comme avant
   // // MG[3] : next mode group from DBB20, as before / groupe de mode suivant depuis DBB20, comme avant
   // // MG[4] : next mode group from DBB20, as before / groupe de mode suivant depuis DBB20, comme avant
   // // MG[5] : next mode group from DBB20, as before / groupe de mode suivant depuis DBB20, comme avant
   // // MG[6] : next mode group from DBB20, as before / groupe de mode suivant depuis DBB20, comme avant
   // // MG[7] : next mode group from DBB20, as before / groupe de mode suivant depuis DBB20, comme avant
   // // MG[8] : next mode group from DBB20, as before / groupe de mode suivant depuis DBB20, comme avant
   // // MG[9] : next mode group from DBB20, as before / groupe de mode suivant depuis DBB20, comme avant
   // // MG[10] : next mode group from DBB20, as before / groupe de mode suivant depuis DBB20, comme avant
END_TYPE
